FUNCTION BytesToString : STRING(1000)
VAR_IN_OUT
	arr : ARRAY[*] OF BYTE;
END_VAR
VAR
	i : DINT;
END_VAR

MEMCPY(ADR(BytesToString), arr, SIZEOF(BytesToString));

END_FUNCTION

(* stored: Version 1.1.0.1, ProductVersion 3.1.4024.11
   POU BytesToString: Id {8f516d69-6ee0-494d-9f37-c28947f679c6}, SpecialFunc None *)
